{attribute 'qualified_only'}
{attribute 'strict'}
TYPE
    T_ExecutionState :
    (
        Ready := 0,
        Starting,
        Busy,
        Aborting
    );
END_TYPE

(* stored: Version 1.1.0.1, ProductVersion 3.1.4024.12
   DUT T_ExecutionState: Id {06db8b1a-766b-063d-044e-a4edc8714d9c} *)
